FUNCTION_BLOCK FB_ATM_Machine IMPLEMENTS I_Machine
VAR_IN_OUT
	xOnButton		:	BOOL;
	xOffButton		:	BOOL;
	xServiceKey		:	BOOL;
	xCardInserted	:	BOOL;
	xCardEjected	:	BOOL;
	xCancelButton	:	BOOL;
END_VAR
VAR_OUTPUT
	ipState	:	I_State	:=	fbOff;
END_VAR
VAR
	fbOff				:	FB_Off(THIS);
	fbIdle				:	FB_Idle(THIS);
	fbMaintenance		:	FB_Maintenance(THIS);
	fbOutOfService		:	FB_OutOfService(THIS);
	fbSelfTest			:	FB_SelfTest(THIS);
	fbServingCustomer	:	FB_ServingCustomer(THIS);
	
	rtrigOnButton		:	R_TRIG;
	rtrigOffButton		:	R_TRIG;
	rtrigCancelButton	:	R_TRIG;
	rtrigCardInserted	:	R_TRIG;
	rtrigCardEjected	:	R_TRIG;
	
	// Simulation Variables
	Sim_TimerTester		:	TON 	:= (PT := T#3S);
	Sim_TimerTransaction:	TON 	:= (PT := T#3S);	
	Sim_xFaultSystem	: 	BOOL;
END_VAR

rtrigOnButton(CLK:= xOnButton);
rtrigOffButton(CLK:= xOffButton);
rtrigCancelButton(CLK:= xCancelButton);
rtrigCardInserted(CLK:= xCardInserted);
rtrigCardEjected(CLK:= xCardEjected);


IF rtrigOnButton.Q THEN
	ipState.Turn_On();
END_IF

IF rtrigOffButton.Q THEN
	ipState.Turn_Off();
END_IF

IF rtrigCancelButton.Q THEN
	ipState.Cancel();
END_IF

IF rtrigCardInserted.Q THEN
	ipState.Card_Inserted();
END_IF

IF rtrigCardEjected.Q THEN
	ipState.Card_Ejected();
END_IF


IF (ipState.Description = E_StateDescription.Idle OR ipState.Description = E_StateDescription.OutOfService) AND xServiceKey THEN
	ipState.Service();
END_IF

IF ipState.Description = E_StateDescription.Maintenance AND NOT xServiceKey THEN
	ipState.Op();
END_IF



// Simulation Variables - Remove and tie to I/O for moving forward
Sim_TimerTester(IN := ipState.Description = E_StateDescription.SelfTest);
IF Sim_TimerTester.Q AND NOT Sim_xFaultSystem THEN
	ipState.SystemTest_OK();
ELSIF Sim_TimerTester.Q  AND Sim_xFaultSystem THEN
	ipState.Failure();
END_IF

Sim_TimerTransaction(IN := ipState.Description = E_StateDescription.ServingCustomer);
IF Sim_TimerTransaction.Q AND NOT Sim_xFaultSystem THEN
	ipState.Card_Ejected();
ELSIF Sim_TimerTransaction.Q AND Sim_xFaultSystem THEN
	ipState.Failure();
END_IF

METHOD FB_Init : BOOL
VAR_INPUT
	(* if TRUE, the retain variables are initialized (warm start / cold start)*)
	bInitRetains	: BOOL;
	(* if TRUE, the instance afterwards gets moved into the copy code (online change)*)
	bInCopyCode	: BOOL;
END_VAR
END_METHOD

PROPERTY IdleState : I_State
GET
IdleState := This^.fbIdle;
END_GET
END_PROPERTY

PROPERTY MaintenanceState : I_State
GET
MaintenanceState := THIS^.fbMaintenance;
END_GET
END_PROPERTY

PROPERTY OffState : I_State
GET
OffState := THIS^.fbOff;
END_GET
END_PROPERTY

PROPERTY OutOfServiceState : I_State
GET
OutOfServiceState := THIS^.fbOutOfService;
END_GET
END_PROPERTY

PROPERTY SelfTestState : I_State
GET
SelfTestState := THIS^.fbSelfTest;
END_GET
END_PROPERTY

PROPERTY ServingCustomerState : I_State
GET
ServingCustomerState := THIS^.fbServingCustomer;
END_GET
END_PROPERTY

METHOD SetState : BOOL
VAR_INPUT
	(* Set the new state to transition*)
	newState	: I_State;
END_VAR
THIS^.ipState := newState;
END_METHOD

END_FUNCTION_BLOCK

(* stored: Version 1.1.0.1, ProductVersion 3.1.4024.12
   POU FB_ATM_Machine: Id {5b7d0fad-4689-0734-192c-cc09349922d8}, SpecialFunc None
   Method FB_Init: Id {ce773053-8282-0701-3e9b-278f6e290085}
   Property IdleState: Id {a1eb420a-8ed4-0616-0e2d-1b421e89e9f7}
   Get Get: Id {e83c7939-15df-076e-27b4-f2de4c103c20}
   Property MaintenanceState: Id {0d2eccca-8fde-0c97-338b-7bf862c57529}
   Get Get: Id {235c7d96-57f5-0fcd-1c86-5da2fca8404d}
   Property OffState: Id {778f5332-0e63-0b0d-3511-d2fbdaaabd9f}
   Get Get: Id {27583678-6dc3-0648-38e2-0d149cf0b76e}
   Property OutOfServiceState: Id {37dde534-1593-0bb3-1839-9b22f775f6ff}
   Get Get: Id {815743aa-9eec-0390-213b-4e51baacdf52}
   Property SelfTestState: Id {f9ba6c6d-bc6a-0ee2-3713-e8984d8cdffd}
   Get Get: Id {a8ca0b12-31d4-042c-2f45-b8bfd007b608}
   Property ServingCustomerState: Id {c17c9037-7517-0bab-3d8f-95edf2b02d76}
   Get Get: Id {0b8858c9-53fc-0334-37d0-d79db04d169b}
   Method SetState: Id {e086c591-e6bf-0cc4-2e48-3fa7b37689a8} *)
